// TIA Portal V19 export
ORGANIZATION_BLOCK "Main"   // OB2701, LAD, ProgramCycle
TITLE = "Main Program Sweep (Cycle)"
// stored: AutoNumber false, IsIECCheckEnabled true, Namespace Unit2.Em6, SetENOAutomatically true
   VAR_INPUT
      Initial_Call : Bool;   // Initial call of this OB
      Remanence : Bool;   // =True, if remanent data are available
   END_VAR
BEGIN

REGION Network 1 (SCL): Call Equipment
   "Unit2.Em6.instSimulation"();

   "Unit2.Em6.CallEquipment_DB"(unitStatus:="Unit2.EmNodes".unitStatus,
                    unitAlarmDB:="Unit2.Alarms".emAlarms[Unit2_EM6],
                    emFeedback:="Unit2.EmNodes".emFeedback[Unit2_EM6]);
END_REGION
END_ORGANIZATION_BLOCK
